// TIA Portal V19 export
FUNCTION "Factora Data Move" : Void   // FC101, STL
{ S7_Optimized_Access := 'TRUE' }
// stored: AutoNumber false
BEGIN

NETWORK
TITLE = Bool Move
      A     "TANK CLEAN";
      =     "Factora Data".STAT0;
      A     "TANK STERILE";
      =     "Factora Data".STAT1;
      A     "R.PROD  AT TANK";

      =     "Factora Data".STAT2;


      A     "Tag_49";
      =     "Factora Data".STAT24;
      A     "FILLER_STERILE";
      =     "Factora Data".STAT25;
      A     "GS22_62";
      =     "Factora Data".STAT26;

NETWORK
TITLE = Word Move
      L     "OP25 TANK".TaStepUpdating;
      T     "Factora Data".STAT16;
      L     "OP25 TANK".TaMainUpdating;
      T     "Factora Data".STAT17;


NETWORK
TITLE = Dword Move
      L     "MeasuredValues".WT0169REAL;
      T     "Factora Data".STAT20;
      L     "Flow Count".Prod_Vol_Count;
      T     "Factora Data".STAT21;

END_FUNCTION
